FUNCTION_BLOCK Picker
VAR_INPUT
    MoveX AT %I* : BOOL;
    MoveY AT %I* : BOOL;
    Rotate AT %I* : BOOL;
    GripRotate AT %I* : BOOL;
END_VAR

END_FUNCTION_BLOCK

(* stored: Version 1.1.0.1, ProductVersion 3.1.4024.10
   POU PICKER: Id {02cfcc68-f3e7-4301-a5c7-ca51bf33dccb}, SpecialFunc None *)
